{attribute 'qualified_only'}
{attribute 'strict'}
{attribute 'to_string'}
TYPE Bedrijfstoestand :
(
	off := 0,
	auto
);
END_TYPE

(* stored: Version 1.1.0.1
   DUT Bedrijfstoestand: Id {0828acc4-c7f1-4b5d-9e19-980aefeb15b9} *)
